{attribute 'GeneratedUsingTerminal: AX8108-0100-0101-0101'}
{attribute addProperty BoxType "AX8108-0100-0101-0101"}
{attribute addProperty Id "FSOEAT %Q*FSOE_BB3344D68"}
{attribute addProperty CRC "1505767614"}
{attribute addProperty Size "8"}
TYPE Standard_Outputdata_59C030BE :
STRUCT
	{attribute addProperty Name "FSOE"}
	FSOE AT %Q* : FSOE_BB3344D6;
END_STRUCT
END_TYPE

(* stored: Version 1.2.0.0, ProductVersion 3.1.4024.9
   DUT Standard_Outputdata_59C030BE: Id {c66b20c3-1a6c-4ddd-8937-eba216274175} *)
